{attribute addProperty BoxType "ER8309-1022-0018"}
{attribute addProperty Id "AI_Inputs_ChannelAT %I*ARRAY[0..1] OF AI_Inputs_Channel_087F71C76480TACHO_Single_Shaft_Mode_Input_Channel_1AT %I*TACHO_Single_Shaft_Mode_Input_Channel_15D41B734860DIG_InputsAT %I*DIG_Inputs_F3F3E4C36480PWM_StatusAT %I*PWM_Status_1DED96921620DEV_InputsAT %I*DEV_Inputs_A68DA3B11620TACHO_Output_Channel_1AT %Q*TACHO_Output_Channel_2290ED3E810DIG_OutputsAT %Q*DIG_Outputs_B71882EA6480PWM_ControlAT %Q*PWM_Control_253BEA613240WcStateAT %I*WcState_F855686C1620InfoDataAT %I*InfoData_BC63D37F80100"}
{attribute addProperty CRC "517518889"}
{attribute addProperty SizeInBites "408"}
{attribute addProperty SizeInBytes "51"}
TYPE ER8309_7EF99CA4 :
STRUCT
	{attribute addProperty Name "AI_Inputs_Channel"}
	AI_Inputs_Channel : ARRAY[0..1] OF AI_Inputs_Channel_087F71C7;
	{attribute addProperty Name "TACHO_Single_Shaft_Mode_Input_Channel_1"}
	TACHO_Single_Shaft_Mode_Input_Channel_1 : TACHO_Single_Shaft_Mode_Input_Channel_15D41B73;
	{attribute addProperty Name "DIG_Inputs"}
	DIG_Inputs : DIG_Inputs_F3F3E4C3;
	{attribute addProperty Name "PWM_Status"}
	PWM_Status : PWM_Status_1DED9692;
	{attribute addProperty Name "DEV_Inputs"}
	DEV_Inputs : DEV_Inputs_A68DA3B1;
	{attribute addProperty Name "TACHO_Output_Channel_1"}
	TACHO_Output_Channel_1 : TACHO_Output_Channel_2290ED3E;
	{attribute addProperty Name "DIG_Outputs"}
	DIG_Outputs : DIG_Outputs_B71882EA;
	{attribute addProperty Name "PWM_Control"}
	PWM_Control : PWM_Control_253BEA61;
	{attribute addProperty Name "WcState"}
	WcState : WcState_F855686C;
	{attribute addProperty Name "InfoData"}
	InfoData : InfoData_BC63D37F;
END_STRUCT
END_TYPE

(* stored: Version 1.2.0.0, ProductVersion 3.1.4024.9
   DUT ER8309_7EF99CA4: Id {95766353-1160-46c5-95ae-fe7482a21d9f} *)
